FUNCTION_BLOCK SawmillControl
  (* Standard: 61499-2 *)
  (* Version 0.1, 2017-00-16, hpea485, UOA *)
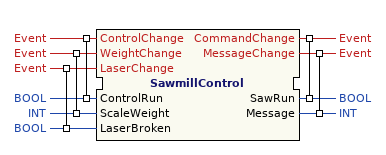
  EVENT_INPUT
    ControlChange WITH ControlRun;
    WeightChange WITH ScaleWeight;
    LaserChange WITH LaserBroken;
  END_EVENT
  EVENT_OUTPUT
    CommandChange WITH SawRun;
    MessageChange WITH Message;
  END_EVENT
  VAR_INPUT
    ControlRun : BOOL;
    ScaleWeight : INT;
    LaserBroken : BOOL;
  END_VAR
  VAR_OUTPUT
    SawRun : BOOL;
    Message : INT;
  END_VAR
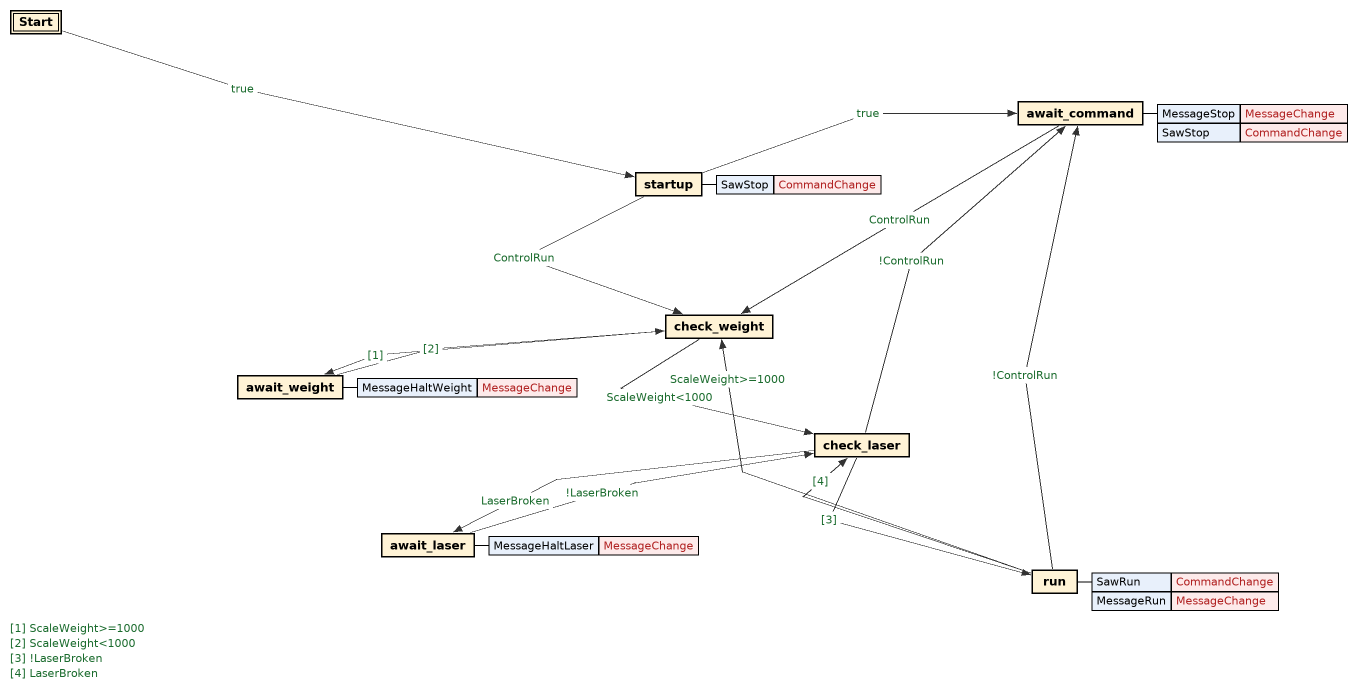
  EC_STATES
    Start;
    startup : SawStop -> CommandChange;
    check_weight;
    check_laser;
    run : SawRun -> CommandChange, MessageRun -> MessageChange;
    await_weight : MessageHaltWeight -> MessageChange;
    await_laser : MessageHaltLaser -> MessageChange;
    await_command : MessageStop -> MessageChange, SawStop -> CommandChange;
  END_STATES
  EC_TRANSITIONS
    Start TO startup := true;
    startup TO check_weight := ControlRun;
    startup TO await_command := true;
    check_weight TO check_laser := ScaleWeight<1000;
    check_weight TO await_weight := ScaleWeight>=1000;
    check_laser TO run := !LaserBroken;
    check_laser TO await_laser := LaserBroken;
    check_laser TO await_command := !ControlRun;
    run TO check_laser := LaserBroken;
    run TO check_weight := ScaleWeight>=1000;
    run TO await_command := !ControlRun;
    await_weight TO check_weight := ScaleWeight<1000;
    await_laser TO check_laser := !LaserBroken;
    await_command TO check_weight := ControlRun;
  END_TRANSITIONS
  ALGORITHM MessageHaltWeight IN C:
me->Message = -1;
  END_ALGORITHM
  ALGORITHM MessageHaltLaser IN C:
me->Message = -2;
  END_ALGORITHM
  ALGORITHM MessageRun IN C:
me->Message = 1;
  END_ALGORITHM
  ALGORITHM MessageStop IN C:
me->Message = 0;
  END_ALGORITHM
  ALGORITHM SawRun IN C:
me->SawRun = 1;
  END_ALGORITHM
  ALGORITHM SawStop IN C:
me->SawRun = 0;
  END_ALGORITHM
END_FUNCTION_BLOCK
